// Mitsubishi GX Works2 project: yes   PLC: Q03UDV

PROGRAM MAIN
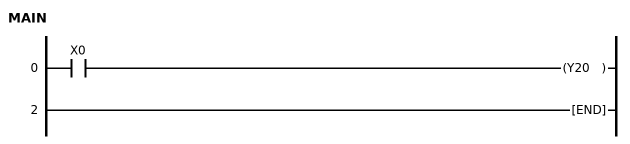
0     LD      X0
      OUT     Y20
2     END
END_PROGRAM
